{attribute 'GeneratedUsingTerminal: AT2000-0233-0022'}
{attribute addProperty BoxType "AT2000-0233-0022"}
{attribute addProperty Id "ControlAT %Q*UINT2Current_setpoint_value_ChAT %Q*ARRAY[0..13] OF INT28"}
{attribute addProperty CRC "2837285957"}
{attribute addProperty Size "30"}
TYPE CC_Outputs_14_Ch_45965511 :
STRUCT
	{attribute addProperty Name "Control"}
	Control AT %Q* : UINT;
	{attribute addProperty Name "Current_setpoint_value_Ch"}
	Current_setpoint_value_Ch AT %Q* : ARRAY[0..13] OF INT;
END_STRUCT
END_TYPE

(* stored: Version 1.2.0.0, ProductVersion 3.1.4024.9
   DUT CC_Outputs_14_Ch_45965511: Id {2ab7ae36-fcb3-4260-b6af-28d66446c68b} *)
